TYPE ST_KashiyamaDryPump EXTENDS ST_RoughPump:
STRUCT

(* Output *)
    //q_xRunDO 	:	BOOL; in Rough PUMP
    {attribute 'pytmc' := '
    pv: RESET_DO;
    field: ZNAM FALSE;
    field: ONAM TRUE;
    io: i
    '}
    q_xResetDo	: 	BOOL;
    {attribute 'pytmc' := '
    pv: LSPD_DO;
    field: ZNAM FALSE;
    field: ONAM TRUE;
    io: i
    '}
    q_xLspdDo	: 	BOOL;
    {attribute 'pytmc' := '
    pv: REM_DO;
    field: ZNAM FALSE;
    field: ONAM TRUE;
    io: i
    '}
    q_xRemoteDo	: 	BOOL;

(* Input *)
{attribute 'pytmc' := '
    pv: REMOTE;
    field: ZNAM FALSE;
    field: ONAM TRUE;
    io: i
    '}
    i_xRemote	:	BOOL;

    {attribute 'pytmc' := '
    pv: ALARM_OK;
    field: ZNAM FALSE;
    field: ONAM TRUE;
    io: i
    '}
    i_xAlarmOK	:	BOOL;
    {attribute 'pytmc' := '
    pv: WARN_OK;
    field: ZNAM FALSE;
    field: ONAM TRUE;
    io: i
    '}
    i_xWarningOK	:	BOOL;
    {attribute 'pytmc' := '
    pv: RUN_DI;
    field: ZNAM FALSE;
    field: ONAM TRUE;
    io: i
    '}
    i_xIsRun		:	BOOL;

(* Logic status *)

    xLspd_IlkENA:   BOOL;

(* EPICS *)
    //xRunSW		:	BOOL; in Rough PUMP
    {attribute 'pytmc' := '
    pv: RESET_SW;
    field: ZNAM FALSE;
    field: ONAM TRUE;
    io: io
    '}
    xResetSW	:	BOOL; //For resetting faults
    {attribute 'pytmc' := '
    pv: LSPD_SW;
    field: ZNAM FALSE;
    field: ONAM TRUE;
    io: io
    '}
    xLspdSW     :   BOOL;
    LowSP  :   REAL := 0.02; //Torr
    HighSP :   REAL; //Torr
    RdyTmr : REAL;
END_STRUCT
END_TYPE

(* stored: Version 1.1.0.1
   DUT ST_KashiyamaDryPump: Id {ea7dbd39-0b45-44ec-97c9-3ee5cc59d920} *)
